Universal Robots PolyScope program: beckon_to_human.urp

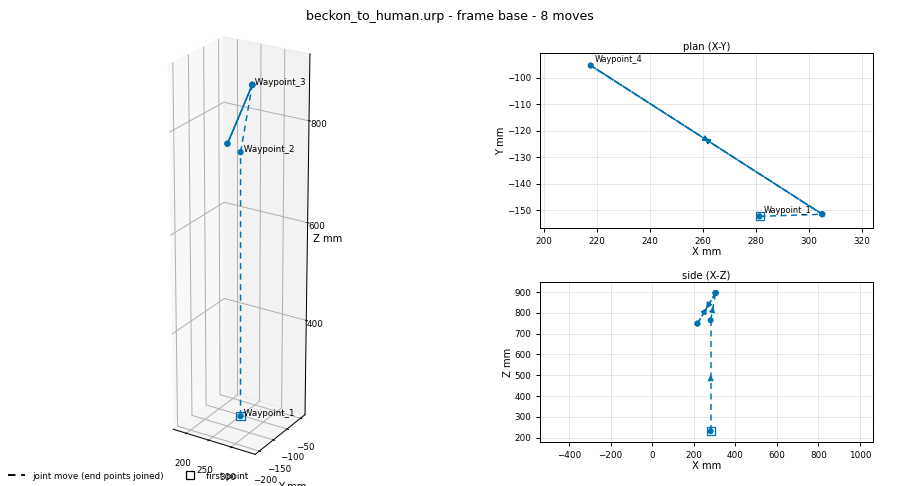
[picture p0: tool path of beckon_to_human.urp in frame base, 8 of 8 moves have a stored position in this frame; points joined in program order, loops and branches not executed]
Program waving (installation=default directory=/home/ur/ursim-current/programs createdIn=3.14.1.1031110 lastSavedIn=3.14.1.1031110 robotSerialNumber=2018309999)
Calibrated DH parameters: a=[0, -0.612, -0.5723, 0, 0, 0]; d=[0.1273, 0, 0, 0.163941, 0.1157, 0.0922]; alpha=[1.570796, 0, 0, 1.570796, -1.570796, 0]; deltaTheta=[0, 0, 0, 0, 0, 0]
Robot Program (runOnlyOnce=false)
  MoveJ speed 60 deg/s, acceleration 80 deg/s^2 (useActiveTCP=true)
    Waypoint Waypoint_1: TCP in base x=281.272 y=-152.342 z=230.789 mm, rx=-0.0012 ry=3.1163 rz=0.0389 rad; joints [1.928, -60.308, -156.017, -52.191, 91.381, 91.901] deg
    Wait Sleep waitTime=3
    Waypoint Waypoint_2: TCP in base x=281.272 y=-152.342 z=764.386 mm, rx=-0.0012 ry=3.1163 rz=0.0389 rad; joints [1.928, -53.484, -102.341, -112.691, 91.381, 91.901] deg
    Waypoint Waypoint_3: motionParameters(jointSpeed=1.047198 jointAcceleration=1.396263 cartesianSpeed=0.25 cartesianAcceleration=1.2); TCP in base x=304.927 y=-151.546 z=895.947 mm, rx=-0.0142 ry=2.1786 rz=0.0643 rad; joints [1.928, -53.484, -102.341, -58.97, 91.381, 91.901] deg
    Wait Sleep waitTime=1
    MoveJ speed 120 deg/s, acceleration 160 deg/s^2 (useActiveTCP=true)
      Waypoint Waypoint_6: TCP in base x=304.927 y=-151.546 z=895.947 mm, rx=-0.0142 ry=2.1786 rz=0.0643 rad; joints [1.928, -53.484, -102.341, -58.97, 91.381, 91.901] deg
      Waypoint Waypoint_4: TCP in base x=217.563 y=-95.429 z=748.543 mm, rx=-1.4129 ry=-1.8003 rz=-0.3603 rad; joints [1.928, -53.484, -100.782, -147.13, 131.627, 155.982] deg
      Waypoint Waypoint_6: TCP in base x=304.927 y=-151.546 z=895.947 mm, rx=-0.0142 ry=2.1786 rz=0.0643 rad; joints [1.928, -53.484, -102.341, -58.97, 91.381, 91.901] deg
      Waypoint Waypoint_4: TCP in base x=217.563 y=-95.429 z=748.543 mm, rx=-1.4129 ry=-1.8003 rz=-0.3603 rad; joints [1.928, -53.484, -100.782, -147.13, 131.627, 155.982] deg
      Waypoint Waypoint_6: TCP in base x=304.927 y=-151.546 z=895.947 mm, rx=-0.0142 ry=2.1786 rz=0.0643 rad; joints [1.928, -53.484, -102.341, -58.97, 91.381, 91.901] deg
    Wait Sleep waitTime=6
